// Mitsubishi GX Works2 project: 230927-002-and   PLC: Q03UDV

// task Task_01 (event TRUE, interval 0, priority 31): POU_01

PROGRAM POU_01
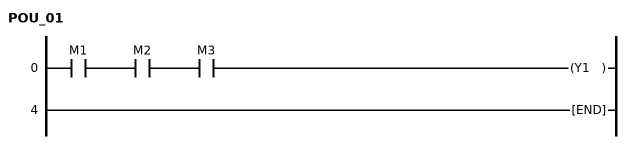
0     LD      M1
      AND     M2
      AND     M3
      OUT     Y1
4     END
END_PROGRAM
